{attribute 'enable_dynamic_creation'}
FUNCTION_BLOCK RecipePoint EXTENDS CloneBase IMPLEMENTS ITF_RecipePoint
VAR
	_xPoint : LREAL;
	_yPoint : LREAL;
	_zPoint : lreal;
END_VAR

METHOD  Clone : ITF_Cloneable
VAR_INPUT
END_VAR
END_METHOD

PROPERTY XPoint : LREAL
GET
XPoint := _xPoint;
END_GET
SET
_xPoint := XPoint;
END_SET
END_PROPERTY

PROPERTY YPoint : LREAL
GET
YPoint := _yPoint;
END_GET
SET
_yPoint := YPoint;
END_SET
END_PROPERTY

PROPERTY ZPoint : LREAL
GET
ZPoint := _zPoint;
END_GET
SET
_zPoint := ZPoint;
END_SET
END_PROPERTY

END_FUNCTION_BLOCK

(* stored: Version 1.1.0.1, ProductVersion 3.1.4024.12
   POU RecipePoint: Id {3eda2ed6-bc47-4b03-a989-037736a4b2eb}, SpecialFunc None
   Method Clone: Id {8bf2e023-210c-4502-b623-bdb8bb439c13}
   Property XPoint: Id {a521519f-84e6-4226-9b89-a54fb8a053a5}
   Get Get: Id {96f679df-201d-4579-80df-b346712a248d}
   Set Set: Id {4ce9243b-c38f-4bfe-a6a0-f048e04a911b}
   Property YPoint: Id {816fed2d-d424-4096-bff3-b7ee3f3ff902}
   Get Get: Id {f8abfc37-a4bf-41f8-9291-ae2127796fe0}
   Set Set: Id {117420c9-2524-4279-971f-6d10eb673264}
   Property ZPoint: Id {c971eefa-6099-42cc-a012-ffa7e14ad24a}
   Get Get: Id {759898a3-f624-4f3b-8067-dd58eed2ecad}
   Set Set: Id {9308dfef-db0f-4510-97bc-978a503d188c} *)
